{attribute 'qualified_only'}
{attribute 'strict'}
{attribute 'to_string'}
TYPE E_LogTransmittal :
(
	invalid := 0,
	toFile,
	viaMQTT,
	viaHTTP,
	viaWS
);
END_TYPE

(* stored: Version 1.1.0.1
   DUT E_LogTransmittal: Id {5f8e71cb-1856-4c45-99b6-4bf2e73e19bc} *)
